PROGRAM POU_StopBladePyP
VAR
END_VAR

GVL_StackBox.bStopBladeA2 := TRUE;
GVL_StackBox.bStopBladeV2 := TRUE;
GVL_StackBox.bStopBladeM2 := TRUE;

END_PROGRAM

(* stored: Version 1.1.0.1, ProductVersion 3.1.4024.12
   POU POU_StopBladePyP: Id {838752ec-6ada-4499-9344-33a85b9aa604}, SpecialFunc None *)
